// TwinCAT 3 PLC project PLC1
// ProgramVersion: 3.1.4024.0
// libraries:
//   Tc2_Standard, * (Beckhoff Automation GmbH)
//   Tc2_System, * (Beckhoff Automation GmbH)
//   Tc3_Module, * (Beckhoff Automation GmbH)
// project tree:
//   / PlcTask.TcTTO
//   POUs/ MAIN.TcPOU
// real-time tasks:
//   TASK PlcTask: cycle T#10ms, priority 20, ADS port 350
// I/O:
//   DEVICE Device 1 (EtherCAT), AmsNetId 10.33.70.115.2.1
//     Term 1 (EK1100) [EK1100 EtherCAT Coupler (2A E-Bus)]
//       Term 2 (EL3058) [EL3058 8Ch. Ana. Input 4-20mA]
//       Term 3 (EL4122) [EL4122 2Ch. Ana. Output  4-20mA, 16bit]
//       Term 4 (EL1008) [EL1008 8Ch. Dig. Input 24V, 3ms]
//       Term 5 (EL7411) [EL7411 BLDC Terminal with incremental encoder/Hall, 50 V DC, 4.5 A]
//       Term 14 (EK1122) [EK1122 2 port EtherCAT junction]
//         Box 15 (EP1111-0000) [EP1111-0000 ID-Switch]
//         Box 16 (EP1008-0001) [EP1008-0001 8 Ch. Dig. Input 24V, 3ms, M8]
//         Box 17 (EP1111-0000) [EP1111-0000 ID-Switch]
//         Box 18 (EP3184-0002) [EP3184-0002 4Ch. Ana. Input +/-10V, 0-10V, 0/4-20mA configurable, single ended]
// variable links:
//   PLC1/PLC1 Instance <-> Device 1 (EtherCAT)/Term 1 (EK1100)/Term 2 (EL3058)
//     PlcTask Inputs/MAIN.AI1 <-> AI Standard Channel 1/Value

CONFIGURATION PLC1
    RESOURCE PLC ON TwinCAT3
        TASK PlcTask(INTERVAL := T#10ms, PRIORITY := 20);
        PROGRAM MAIN WITH PlcTask : MAIN;
    END_RESOURCE
END_CONFIGURATION

// ---- POUs/MAIN.TcPOU
PROGRAM MAIN
VAR
	
	AI1 AT %I* : INT;
	AIs AT %I* : MDP5001_300_EE3A5F5D;
	AIsCh AT %I* : MDP5001_300_4B3D2459;
END_VAR

END_PROGRAM
